PROGRAM MAIN
VAR
	AxisPowTestSuite : AxisPowerTestSuite;
END_VAR

AxisPowTestSuite();

END_PROGRAM

(* stored: Version 1.1.0.1
   POU MAIN: Id {4c2acc94-7e0b-4045-bc96-4e57a86837e2}, SpecialFunc None *)
